// Mitsubishi GX Works2 project: DZRN_DDRVA_runStep   PLC: FX3U/FX3UC

PROGRAM MAIN
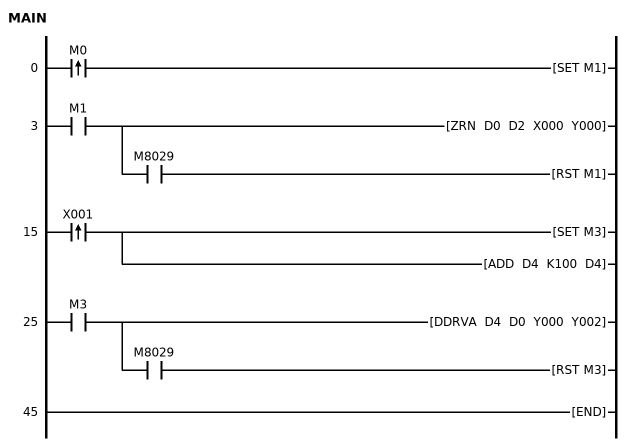
0     LDP     M0
      SET     M1
3     LD      M1
      ZRN     D0 D2 X000 Y000
      AND     M8029
      RST     M1
15    LDP     X001
      SET     M3
      ADD     D4 K100 D4
25    LD      M3
      DDRVA   D4 D0 Y000 Y002
      AND     M8029
      RST     M3
45    END
END_PROGRAM
